Fanuc KAREL source: kt00151.KL

-- PROVISIONAL review KL for V770-1; original PC SHA256 bf37a5ee10efe01aa74d675af6250f9aa140814d970e1f9addaac028faf0677f
-- Incomplete behavior may be omitted. Consult companion uncertainty JSON. Do not deploy.
PROGRAM KT00151
%NOLOCKGROUP
VAR
  OUT : INTEGER
-- UNRESOLVED_DECL Y1 type=002018
-- UNRESOLVED_DECL H2 type=002017
BEGIN
  -- UNRESOLVED_PC offsets 5-19; opcodes 2E,22,9D,33,B2
  -- UNRESOLVED_PC offsets 24-38; opcodes 2E,22,9D,33,B4
  -- UNRESOLVED_PC offsets 43-68; opcodes 22,9D,33,B1,22,9D,33,B3,55,23
  -- UNRESOLVED_PC offsets 73-77; opcodes 7F
END KT00151
